{attribute 'qualified_only'}
VAR_GLOBAL PERSISTENT
	
stPartsInspection			: ST_PartsInspection;
stUserLogHMI				: ARRAY[0..250] OF ST_UserLogHMI;
UserId						: UINT;
ast_i28LasResult            : ARRAY [0..250] OF st_i28LasResult;
nLeakTestID					: UINT;

nCycleNumber				: INT;
	
END_VAR

(* stored: Version 1.1.0.1, ProductVersion 3.1.4024.13
   GVL GVL_PERSIST: Id {d7074b9f-b8f7-43b8-b977-625646657a49} *)
